FUNCTION_BLOCK RingCriticalSection2 (* Basic Function Block Type *)
  (* Standard: 61499-2 *)
  (* Version 0.2, 2003-12-04, JHC, Rockwell Automation, Renamed for better indexing. *)
  (* Version 0.1, 2002-11-05, JHC, Rockwell Automation, Corrected missing ST element in Algorithm REQ. *)
  (* Version 0.0, 2000-05-30, JHC, Rockwell Automation *)
  (* Compiler header: package fb.rt.cs725; *)
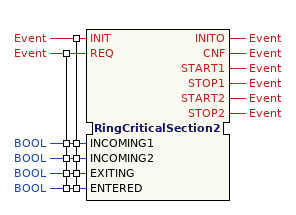
  EVENT_INPUT
    INIT WITH INCOMING1, INCOMING2, EXITING, ENTERED; (* Initialization Request *)
    REQ WITH INCOMING1, INCOMING2, EXITING, ENTERED; (* Normal Execution Request *)
  END_EVENT
  EVENT_OUTPUT
    INITO; (* Initialization Confirm *)
    CNF; (* Execution Confirmation *)
    START1;
    STOP1;
    START2;
    STOP2;
  END_EVENT
  VAR_INPUT
    INCOMING1 : BOOL; (* Input event qualifier *)
    INCOMING2 : BOOL;
    EXITING : BOOL;
    ENTERED : BOOL;
  END_VAR
  VAR
    TOKEN_CLIENT : BOOL;
    TOKEN_BLOCK : BOOL;
  END_VAR
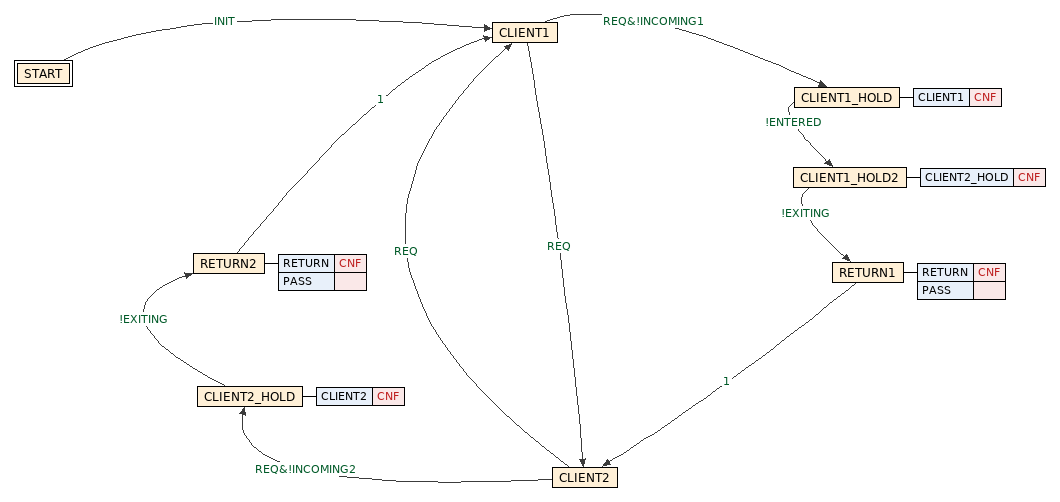
  EC_STATES
    START; (* Initial State *)
    CLIENT1;
    CLIENT1_HOLD : CLIENT1 -> CNF;
    CLIENT1_HOLD2 : CLIENT2_HOLD -> CNF;
    RETURN1 : RETURN -> CNF, PASS;
    CLIENT2;
    CLIENT2_HOLD : CLIENT2 -> CNF;
    RETURN2 : RETURN -> CNF, PASS;
  END_STATES
  EC_TRANSITIONS
    CLIENT1 TO CLIENT1_HOLD := REQ&!INCOMING1;
    START TO CLIENT1 := INIT;
    CLIENT1_HOLD TO CLIENT1_HOLD2 := !ENTERED;
    CLIENT1_HOLD2 TO RETURN1 := !EXITING;
    RETURN1 TO CLIENT2 := 1;
    CLIENT2 TO CLIENT2_HOLD := REQ&!INCOMING2;
    CLIENT2_HOLD TO RETURN2 := !EXITING;
    RETURN2 TO CLIENT1 := 1;
    CLIENT2 TO CLIENT1 := REQ;
    CLIENT1 TO CLIENT2 := REQ;
  END_TRANSITIONS
  ALGORITHM INIT IN ST: (* Initialization algorithm *)
TOKEN_BLOCK := FALSE;
TOKEN_CLIENT := FALSE;
  END_ALGORITHM
  ALGORITHM PASS IN ST: (* Normally executed algorithm *)
IF TOKEN_CLIENT THEN
TOKEN_CLIENT := FALSE;
ELSE
TOKEN_CLIENT := TRUE;
END_IF
  END_ALGORITHM
  ALGORITHM CLIENT1 IN ST:
System.out.println(">>>>    CLIENT ONE HAS CRITICAL SECTION");
TOKEN_BLOCK := TRUE;
START1.serviceEvent(this);
STOP2.serviceEvent(this);
  END_ALGORITHM
  ALGORITHM CLIENT2 IN ST:
System.out.println(">>>>    CLIENT TWO HAS CRITICAL SECTION");
TOKEN_BLOCK := TRUE;
STOP1.serviceEvent(this);
START2.serviceEvent(this);
  END_ALGORITHM
  ALGORITHM RETURN IN ST:
System.out.println(">>>>    EXITING CRITICAL SECTION");
TOKEN_BLOCK := FALSE;
START1.serviceEvent(this);
START2.serviceEvent(this);
  END_ALGORITHM
  ALGORITHM CLIENT1_HOLD IN ST:
System.out.println(">>>>    CLIENT ONE_HOLD");
STOP2.serviceEvent(this);
  END_ALGORITHM
  ALGORITHM CLIENT2_HOLD IN ST:
System.out.println(">>>>    CLIENT TWO_HOLD");
STOP1.serviceEvent(this);
  END_ALGORITHM
END_FUNCTION_BLOCK
